FUNCTION_BLOCK PUBLIC FB_DATETIME
VAR_INPUT
END_VAR
VAR_OUTPUT
END_VAR
VAR
END_VAR

METHOD PUBLIC GetCurrentDateTime : DT
VAR_INPUT
END_VAR
VAR
	SystemTime    : GETSYSTEMTIME;
	timeAsFileTime  : T_FILETIME;
	timeAsDT        : DT;
END_VAR
SystemTime( timeLoDW =>timeAsFileTime.dwLowDateTime , timeHiDW =>timeAsFileTime.dwHighDateTime );
GetCurrentDateTime := FILETIME_TO_DT( timeAsFileTime );
END_METHOD

METHOD PUBLIC GetTimeDiff : TIME
VAR_INPUT
	In1 : TIME;
	In2 : TIME;
END_VAR
GetTimeDiff := In2 - In1;
END_METHOD

METHOD PUBLIC GetTimeSince : TIME
VAR_INPUT
	In : TIME;
END_VAR
GetTimeSince := TIME() - In;
END_METHOD

END_FUNCTION_BLOCK

(* stored: Version 1.1.0.1, ProductVersion 3.1.4024.12
   POU FB_DATETIME: Id {c45fc1db-f5ef-46e9-83f3-709ac35ac1a8}, SpecialFunc None
   Method GetCurrentDateTime: Id {a443d8eb-2ec5-4fa1-887d-ccfaf4d9e3a8}
   Method GetTimeDiff: Id {a91b3ef1-003e-431e-a9e9-71c26a60e592}
   Method GetTimeSince: Id {97f2aa0c-de9a-4816-bae2-a100c339d20e} *)
